{attribute 'pack_mode' := '0'}
TYPE CyltronicProcessDataOutActual :
STRUCT
	MotionMode 			 : CyltronicMotionMode;
	TargetPosition 		 : REAL;
	SpeedOverride 		 : USINT;
	ForceOverride 		 : USINT;
	AccelerationOverride : USINT;
END_STRUCT
END_TYPE

(* stored: Version 1.1.0.1, ProductVersion 3.1.4024.10
   DUT CyltronicProcessDataOutActual: Id {d7e7a496-5346-4b2d-98ee-99c7a434bdba} *)
